  FT_SEARCH_ACC=0.5
  FT_SEARCH_ANG_SPD=3.0
  FT_SEARCH_ANG_ACC=10.0
  FT_SEARCH_RETRACT_ACC=10.0
  FT_SEARCH_RETRACT_SPD=3.0
  FT_SEARCH_RETRACT_M=0.002
  FT_SEARCH_RETRACT_RAD=d2r(4.25)
  ft_search_history_cntr=0
  def ft_trajectory_search_start(f3d=-1.0,t3d=-1.0):
  ft_select=ON_FALSE8D
  ft_limits=ON_ZERO8D
  ft_abs=ON_FALSE6D
  frameID=0
  frameRPY=ON_ZERO3D
  popupmsg=False
  speedLimit=0
  if(f3d>0):
  ft_select[6]=True
  ft_limits[6]=f3d
  end
  if(t3d>0):
  ft_select[7]=True
  ft_limits[7]=t3d
  end
  retVal=ft_limit_start(ft_select,ft_limits,ft_abs,speedLimit,frameID,frameRPY,popupmsg)
  cb_trajectory_return_validator(retVal,"F/T Limit: ")
  return retVal
  end
  def ft_trajectory_limited(trajectoryID,ft_select=ON_FALSE8D,ft_limits=ON_ZERO8D,ft_abs=ON_FALSE6D,frameID=0,frameRPY=ON_ZERO3D,isSearchReturn=False,popupmsg=True):
  speedLimit=0
  retVal=ft_limit_start(ft_select,ft_limits,ft_abs,speedLimit,frameID,frameRPY,popupmsg)
  cb_trajectory_return_validator(retVal,"F/T Limit: ")
  retVal=cb_trajectory(trajectoryID,isSearchReturn,popupmsg)
  ft_limit_stop()
  return retVal
  end
  def ft_trajectory_move_relative_limited_array(relativeOffsetsPoseArray=[ON_ZEROPOSE],ft_select=ON_FALSE8D,ft_limits=ON_ZERO8D,ft_abs=ON_FALSE6D,frameID=1,frameRPY=ON_ZERO3D,speed=0.05,acc=1.2,angularSpeed=3.0,angularAcc=10.0,isSearchReturn=False,popupmsg=True):
  local retVal=0
  frameRotVec=rpy2rotvec(frameRPY)
  frame6D=[0.0,0.0,0.0,frameRotVec[0],frameRotVec[1],frameRotVec[2]]
  frame=p[0.0,0.0,0.0,frameRotVec[0],frameRotVec[1],frameRotVec[2]]
  if((frameID%2)==1):
  startPose=get_actual_tcp_pose()
  startPose=pose_trans(startPose,frame)
  else:
  startPose=pose_trans(ON_ZEROPOSE,frame)
  end
  cb_trajectory_path_init(True,frameID,frame6D,speed,acc,angularSpeed,angularAcc)
  retVal=on_xmlrpc.cb_trajectory_waypoint([startPose[0]*1000.0,startPose[1]*1000.0,startPose[2]*1000.0,startPose[3],startPose[4],startPose[5]])
  cb_trajectory_return_validator(retVal,"OnWaypoint: ")
  cb_trajectory_waypoints_init(relativeOffsetsPoseArray,startPose,True,frameID)
  trajectoryID=cb_trajectory_path_init_end()
  retVal=ft_trajectory_limited(trajectoryID,ft_select,ft_limits,ft_abs,frameID,frameRPY,isSearchReturn,popupmsg)
  return retVal
  end
  def ft_trajectory_move_relative_limited(relativeOffsets=ON_ZEROPOSE,ft_select=ON_FALSE8D,ft_limits=ON_ZERO8D,ft_abs=ON_FALSE6D,frameID=1,frameRPY=ON_ZERO3D,speed=0.05,acc=1.2,angularSpeed=3.0,angularAcc=10.0,isSearchReturn=False,popupmsg=True):
  retVal=ft_trajectory_move_relative_limited_array([relativeOffsets],ft_select,ft_limits,ft_abs,frameID,frameRPY,speed,acc,angularSpeed,angularAcc,isSearchReturn,popupmsg)
  return retVal
  end
  def ft_trajectory_move_absolute_limited_array(fixPoseArray,ft_select=ON_FALSE8D,ft_limits=ON_ZERO8D,ft_abs=ON_FALSE6D,speed=0.05,acc=1.2,angularSpeed=3.0,angularAcc=10.0,isSearchReturn=False,popupmsg=True):
  local retVal=0
  frame6D=ON_ZERO6D
  frameID=0
  frameRPY=ON_ZERO3D
  local startPose=ON_ZEROPOSE
  cb_trajectory_path_init(False,frameID,frame6D,speed,acc,angularSpeed,angularAcc)
  cb_trajectory_waypoints_init(fixPoseArray,startPose,False,frameID)
  trajectoryID=cb_trajectory_path_init_end()
  retVal=ft_trajectory_limited(trajectoryID,ft_select,ft_limits,ft_abs,frameID,frameRPY,isSearchReturn,popupmsg)
  return retVal
  end
  def ft_trajectory_move_absolute_limited(fixPose,ft_select=ON_FALSE8D,ft_limits=ON_ZERO8D,ft_abs=ON_FALSE6D,speed=0.05,acc=1.2,angularSpeed=3.0,angularAcc=10.0,isSearchReturn=False,popupmsg=True):
  retVal=ft_trajectory_move_absolute_limited_array([fixPose],ft_select,ft_limits,ft_abs,speed,acc,angularSpeed,angularAcc,isSearchReturn,popupmsg)
  return retVal
  end
  def ft_search_relativeZ(tool_index,searchDistZ,speed=0.03,forceZ=5.0,popupmsg=True):
  on_tcp_set_actual_to(tool_index!=ON_DI_SECONDARY)
  ft_select=ON_FALSE8D
  ft_select[2]=True
  ft_limits=ON_ZERO8D
  ft_limits[2]=forceZ
  ft_abs=ON_FALSE6D
  frameID=1
  frameRPY=ON_ZERO3D
  searchUntil=ON_ZEROPOSE
  searchUntil[2]=searchDistZ
  isSearchReturn=True
  local retVal=ft_trajectory_move_relative_limited(searchUntil,ft_select,ft_limits,ft_abs,frameID,frameRPY,speed,FT_SEARCH_ACC,FT_SEARCH_ANG_SPD,FT_SEARCH_ANG_ACC,isSearchReturn,popupmsg)
  return retVal
  end
  def ft_search_get_retract_pose(poseArray,actualStep,retract_m=-1,retract_rad=-1):
  local SafeIndex=actualStep+1
  if SafeIndex>=FT_SEARCH_HISTORY_LENGTH:
  SafeIndex=0
  end
  local actualPose=poseArray[actualStep]
  local safePose=poseArray[SafeIndex]
  local directionPose=pose_trans(pose_inv(actualPose),safePose)
  local directionUnit=normalize([directionPose[0],directionPose[1],directionPose[2],directionPose[3],directionPose[4],directionPose[5]])
  local Pdist=pose_dist(actualPose,safePose)
  local retractVector=directionPose
  if(retract_m>=0):
  retractVector[0]=directionUnit[0]*retract_m
  retractVector[1]=directionUnit[1]*retract_m
  retractVector[2]=directionUnit[2]*retract_m
  end
  if(retract_rad>=0):
  retractVector[3]=directionUnit[3]*retract_rad
  retractVector[4]=directionUnit[4]*retract_rad
  retractVector[5]=directionUnit[5]*retract_rad
  end
  ft_search_safe_pose=pose_trans(actualPose,retractVector)
  return ft_search_safe_pose
  end
  thread ft_search_safety_thread():
  ft_search_abscntr=0
  ft_search_history_cntr=0
  while True:
  enter_critical
  ft_search_abscntr=ft_search_abscntr+1
  ft_search_history_cntr=ft_search_history_cntr+1
  if ft_search_history_cntr>=FT_SEARCH_HISTORY_LENGTH:
  ft_search_history_cntr=0
  end
  ft_search_history[ft_search_history_cntr]=get_actual_tcp_pose()
  exit_critical
  sync()
  end
  end
  ft_search_safety_thrd=run ft_search_safety_thread()
  def ft_search_retract(retractPose):
  if(on_speedl_integer_get()==0):
  movel(retractPose,a=FT_SEARCH_ACC,v=FT_SEARCH_RETRACT_SPD)
  else:
  cb_trajectory_move_absolute(retractPose,FT_SEARCH_RETRACT_SPD,FT_SEARCH_ACC,(FT_SEARCH_RETRACT_SPD*4.0),(FT_SEARCH_ACC*4.0),False)
  end
  end
  def ft_search_OK_retract(retractPose):
  if ft_search_return==0:
  ft_search_retract(retractPose)
  end
  end

  #======    End of OnRobot FT Trajectory    ======#
  #======    OnRobot FT Trajectory Spiral    ======#

  def cb_trajectory_spiral(spiralStartEndPoses=[ON_ZEROPOSE,ON_ZEROPOSE],isRelative=True,speed=0.05,acc=1.2,angularSpeed=3.0,angularAcc=10.0,increase=0.001,direction=False,closingCircle=False,popupmsg=True):
  local retVal=0
  local isSearchReturn=False
  trajectoryID=cb_trajectory_spiral_init(spiralStartEndPoses,isRelative,speed,acc,angularSpeed,angularAcc,increase,direction,closingCircle)
  retVal=cb_trajectory(trajectoryID,isSearchReturn,popupmsg)
  return retVal
  end
  def cb_trajectory_spiral_limited(spiralStartEndPoses=[ON_ZEROPOSE,ON_ZEROPOSE],ft_select=ON_FALSE8D,ft_limits=ON_ZERO8D,ft_abs=ON_FALSE6D,isRelative=True,speed=0.05,acc=1.2,angularSpeed=3.0,angularAcc=10.0,increase=0.01,direction=False,closingCircle=False,isSearchReturn=False,popupmsg=True):
  local retVal=0
  local frameRPY=ON_ZERO3D
  local frameID=1
  trajectoryID=cb_trajectory_spiral_init(spiralStartEndPoses,isRelative,speed,acc,angularSpeed,angularAcc,increase,direction,closingCircle)
  retVal=ft_trajectory_limited(trajectoryID,ft_select,ft_limits,ft_abs,frameID,frameRPY,isSearchReturn,popupmsg)
  return retVal
  end

  #======    End of OnRobot FT Trajectory Spiral    ======#
  #======    OnRobot FT Insert Part Messages    ======#

  ft_insert_part_error_title="OnRobot - Insert Part error"
  ft_insert_part_state_error_start="Wrong F/T Insert Part status when initializing.<br>Another thread is using an F/T Insert Part command. Program halted."
  ft_insert_part_state_error_return="Wrong F/T Insert Part status when returning.<br>Another thread is using an F/T Insert Part command. Program halted."
  ft_insert_part_return_title="OnRobot - Insert Part"
  ft_insert_part_return_0="The insertion has reached the maximal insertion depth."
  ft_insert_part_return_1="The insertion bumped after the minimal insertion depth."
  ft_insert_part_return_2="The insertion slowed down after the minimal insertion depth."
  ft_insert_part_return_3="The insertion got stuck before the minimal insertion depth."
  ft_insert_part_return_4="The command has timed out after the minimal insertion depth."
  ft_insert_part_return_5="The command has timed out before the minimal insertion depth."
  ft_insert_part_return_6="The side-force/-torque limit has been reached after the minimal insertion depth."
  ft_insert_part_return_7="The side-force/-torque limit has been reached before the minimal insertion depth."
  ft_insert_part_return_8="Parameter error returned from the Compute Box.<br>Check the parameters for the F/T Insert Part command."
  ft_insert_part_return_unknown="F/T Insert Part finished with unknown return value."

  #======    End of OnRobot FT Insert Part Messages    ======#
  #======    OnRobot FT Insert Part    ======#

  ft_insert_part_state=0
  ft_insert_part_return=0
  ft_sensor_filter_insertpart_hex=6
  ft_insert_part_frameID=1
  ft_insert_part_frameID_default=1
  ft_insert_part_frameRPY=ON_ZERO3D
  ft_insert_part_frameRPY_default=ON_ZERO3D
  ft_insert_part_retAccept=[True,True,True,False,False,False,False,False,False]
  ft_insert_part_retAccept_default=[True,True,True,False,False,False,False,False,False]
  FT_INSERT_PART_STATE_IDLE=0
  FT_INSERT_PART_STATE_INIT=1
  FT_INSERT_PART_STATE_STARTED=2
  FT_INSERT_PART_STATE_RETURNING=3
  ft__insert_part_param_error_minDistZ="Please define parameter 'minDistZ' as a positive real number in meters!"
  ft__insert_part_param_error_forceZ="Please define parameter 'forceZ' as a positive number in Newtons!"
  ft__insert_part_param_error_maxDistZ="Please define parameter 'maxDistZ' as a positive real number in meters!"
  ft__insert_part_param_error_maxDistZ_minDistZ="Please define the parameters as 'maxDistZ' >= 'minDistZ'!"
  ft__insert_part_param_error_expSpeed="Please define parameter 'expSpeed' as a positive real number in meters!"
  ft__insert_part_param_error_deltaForce="Please define parameter 'deltaForce' as a positive number in Newtons!"
  ft__insert_part_param_error_timeOut="Please define parameter 'timeOut' as a positive number in seconds!"
  ft__insert_part_param_error_FTLimits="Please define parameter 'FTLimits' as a 6-element array of positive numbers in Newtons & Newton-meters!"
  ft__insert_part_param_error_PGainFxy="Please define parameter 'PGainFxy' as a positive real number!"
  ft__insert_part_param_error_PGainFz="Please define parameter 'PGainFz' as a positive real number!"
  ft__insert_part_param_error_PGainTxy="Please define parameter 'PGainTxy' as a positive real number!"
  ft__insert_part_param_error_PGainTz="Please define parameter 'PGainTz' as a positive real number!"
  def ft_insert_part(forceZ,minDistZ,maxDistZ=0.0,deltaForce=0.0,expSpeed=0.0,timeOut=0,compliance=[True,True,True,True,True,True],FTLimits=ON_ZERO6D,PGainFxy=1.0,PGainFz=1.0,PGainTxy=0.2,PGainTz=0.2,popupmsg=True):
  sync()
  if ON_DEBUG_LOG:
  textmsg("Insert Part starting..")
  end
  if not(ft_insert_part_state==FT_INSERT_PART_STATE_IDLE):
  textmsg("ft_insert_part_state: ",ft_insert_part_state)
  popup(ft_insert_part_state_error_start,title=ft_insert_part_error_title,error=True,blocking=False)
  halt
  else:
  enter_critical
  ft_insert_part_state=FT_INSERT_PART_STATE_INIT
  exit_critical
  end
  ft_insert_part_return=0
  if not(minDistZ>=0):
  ft_insert_part_return=8
  popup(ft__insert_part_param_error_minDistZ,title=ft_insert_part_error_title,error=True,blocking=True)
  elif not(forceZ!=0):
  ft_insert_part_return=8
  popup(ft__insert_part_param_error_forceZ,title=ft_insert_part_error_title,error=True,blocking=True)
  elif not(maxDistZ>=0):
  ft_insert_part_return=8
  popup(ft__insert_part_param_error_maxDistZ,title=ft_insert_part_error_title,error=True,blocking=False)
  elif not(maxDistZ>=minDistZ or maxDistZ==0):
  ft_insert_part_return=8
  popup(ft__insert_part_param_error_maxDistZ_minDistZ,title=ft_insert_part_error_title,error=True,blocking=False)
  elif not(expSpeed>=0):
  ft_insert_part_return=8
  popup(ft__insert_part_param_error_expSpeed,title=ft_insert_part_error_title,error=True,blocking=False)
  elif not(deltaForce>=0):
  ft_insert_part_return=8
  popup(ft__insert_part_param_error_deltaForce,title=ft_insert_part_error_title,error=True,blocking=False)
  elif not(timeOut>=0):
  ft_insert_part_return=8
  popup(ft__insert_part_param_error_timeOut,title=ft_insert_part_error_title,error=True,blocking=False)
  elif not(FTLimits[0]>=0):
  ft_insert_part_return=8
  popup(ft__insert_part_param_error_FTLimits,title=ft_insert_part_error_title,error=True,blocking=False)
  elif not(FTLimits[1]>=0):
  ft_insert_part_return=8
  popup(ft__insert_part_param_error_FTLimits,title=ft_insert_part_error_title,error=True,blocking=False)
  elif not(FTLimits[3]>=0):
  ft_insert_part_return=8
  popup(ft__insert_part_param_error_FTLimits,title=ft_insert_part_error_title,error=True,blocking=False)
  elif not(FTLimits[4]>=0):
  ft_insert_part_return=8
  popup(ft__insert_part_param_error_FTLimits,title=ft_insert_part_error_title,error=True,blocking=False)
  elif not(FTLimits[5]>=0):
  ft_insert_part_return=8
  popup(ft__insert_part_param_error_FTLimits,title=ft_insert_part_error_title,error=True,blocking=False)
  elif not(PGainFxy>0):
  ft_insert_part_return=8
  popup(ft__insert_part_param_error_PGainFxy,title=ft_insert_part_error_title,error=True,blocking=False)
  elif not(PGainFz>0):
  ft_insert_part_return=8
  popup(ft__insert_part_param_error_PGainFz,title=ft_insert_part_error_title,error=True,blocking=False)
  elif not(PGainTxy>0):
  ft_insert_part_return=8
  popup(ft__insert_part_param_error_PGainTxy,title=ft_insert_part_error_title,error=True,blocking=False)
  elif not(PGainTz>0):
  ft_insert_part_return=8
  popup(ft__insert_part_param_error_PGainTz,title=ft_insert_part_error_title,error=True,blocking=False)
  end
  if(ft_insert_part_return!=0):
  halt
  end
  on_tcp_offset_send(get_tcp_offset())
  local retAccept=ft_insert_part_retAccept
  ft_insert_part_retAccept=ft_insert_part_retAccept_default
  local ft_compliance=compliance
  ft_compliance[2]=True
  local ft_threshold=[FTLimits[0],FTLimits[1],(forceZ+deltaForce),FTLimits[3],FTLimits[4],FTLimits[5]]
  i=0
  while i<6:
  if ft_compliance[i]:
  ft_threshold[i]=0
  end
  i=i+1
  end
  local flags=binary_list_to_integer(ft_compliance)+(ft_insert_part_frameID*64)
  ft_insert_part_frameID=ft_insert_part_frameID_default
  local ft_insert_part_frame=rpy2rotvec(ft_insert_part_frameRPY)
  ft_insert_part_frameRPY=ft_insert_part_frameRPY_default
  sync()
  ft_insert_part_return=ft_pin_insertion(minDistZ,forceZ,compliance,maxDistZ,expSpeed,deltaForce,timeOut,FTLimits,PGainFxy,PGainFz,PGainTxy,PGainTz)
  if ON_DEBUG_LOG:
  textmsg("Insert Part returned.")
  end
  if ft_insert_part_return==0:
  if(popupmsg and(not retAccept[0])):
  popup(ft_insert_part_return_0,title=ft_insert_part_return_title,warning=True,blocking=True)
  end
  elif ft_insert_part_return==1:
  if(popupmsg and(not retAccept[1])):
  popup(ft_insert_part_return_1,title=ft_insert_part_return_title,warning=True,blocking=True)
  end
  elif ft_insert_part_return==2:
  if(popupmsg and(not retAccept[2])):
  popup(ft_insert_part_return_2,title=ft_insert_part_return_title,warning=True,blocking=True)
  end
  elif ft_insert_part_return==3:
  if(popupmsg and(not retAccept[3])):
  popup(ft_insert_part_return_3,title=ft_insert_part_return_title,warning=True,blocking=True)
  end
  elif ft_insert_part_return==4:
  if(popupmsg and(not retAccept[4])):
  popup(ft_insert_part_return_4,title=ft_insert_part_return_title,warning=True,blocking=True)
  end
  elif ft_insert_part_return==5:
  if(popupmsg and(not retAccept[5])):
  popup(ft_insert_part_return_5,title=ft_insert_part_return_title,warning=True,blocking=True)
  end
  elif ft_insert_part_return==6:
  if(popupmsg and(not retAccept[6])):
  popup(ft_insert_part_return_6,title=ft_insert_part_return_title,warning=True,blocking=True)
  end
  elif ft_insert_part_return==7:
  if(popupmsg and(not retAccept[7])):
  popup(ft_insert_part_return_7,title=ft_insert_part_return_title,warning=True,blocking=True)
  end
  else:
  popup(ft_insert_part_return_unknown,title=ft_insert_part_return_title,warning=True,blocking=True)
  end
  enter_critical
  ft_insert_part_state=FT_INSERT_PART_STATE_IDLE
  exit_critical
  if ON_DEBUG_LOG:
  textmsg("End of Insert Part.")
  end
  return ft_insert_part_return
  end
  ft_peakFzScanner_flag=False
  ft_abs_Fz=0
  ft_abs0_Fz=False
  thread ft_peakFzScanner():
  ft_peakFzScanner_flag=True
  ft_abs_Fz=0
  while(ft_peakFzScanner_flag==True):
  local norm_Fz=norm(FT_Tool[2])
  if(ft_abs0_Fz):
  ft_abs_Fz=0
  ft_abs0_Fz=False
  elif(ft_abs_Fz<norm_Fz):
  ft_abs_Fz=norm_Fz
  end
  sync()
  end
  end
  ft_fpid_i_pin=0.0
  ft_fpid_d_pin=0.0
  ft_fpid_i_pin_default=0.0
  ft_fpid_d_pin_default=0.0
  ft_tpid_i_pin=0.0
  ft_tpid_d_pin=0.0
  ft_tpid_i_pin_default=0.0
  ft_tpid_d_pin_default=0.0
  def ft_pin_insertion(minDistZ,forceZ,compliance=[True,True,True,True,True,True],maxDistZ=0,expSpeed=0,deltaForce=1,timeOut=0,FTLimits=[999,999,0,999,999,999],PGainFxy=1.0,PGainFz=1.0,PGainTxy=0.2,PGainTz=0.2):
  sync()
  local pinRet=0
  local frameID=1
  local startPose=get_actual_tcp_pose()
  if maxDistZ==0:
  maxDistZ=minDistZ
  end
  local dist2Reach=maxDistZ
  sync()
  local selectThreshold=[False,False,False,False,False,False]
  local ft_select=compliance
  ft_select[2]=True
  local ft_values=[0.0,0.0,0.0,0.0,0.0,0.0]
  ft_values[2]=forceZ+0.0
  local i=0
  while(i<6):
  selectThreshold[i]=not(ft_select[i])
  i=i+1
  end
  local pin_useTimeOut=True
  if timeOut==0:
  pin_useTimeOut=False
  end
  local timeOut100ms=timeOut*10
  local deltaD=expSpeed/10
  ft_pin_currentDist=0
  local peakScanner=run ft_peakFzScanner()
  sync()
  local pin_gainP=[PGainFxy,PGainFxy,PGainFz,PGainTxy,PGainTxy,PGainTz]
  local pin_gainI=[ft_fpid_i_pin,ft_fpid_i_pin,ft_fpid_i_pin,ft_tpid_i_pin,ft_tpid_i_pin,ft_tpid_i_pin]
  local pin_gainD=[ft_fpid_d_pin,ft_fpid_d_pin,ft_fpid_d_pin,ft_tpid_d_pin,ft_tpid_d_pin,ft_tpid_d_pin]
  if on_hex:
  on_xmlrpc.ft_sensor_filter(ft_sensor_filter_insertpart_hex)
  end
  pin_speed_variation=0.0
  pin_keep_force=-1.0
  pin_auto_keep_force=False
  pin_keep_torque=-1.0
  pin_auto_keep_torque=False
  ft_ftcontrol_start(ft_select=ft_select,ft_values=ft_values,frameID=frameID,frameRPY=[0,0,0],gainP=pin_gainP,gainI=pin_gainI,gainD=pin_gainD,speed_variation=pin_speed_variation,keep_force=pin_keep_force,auto_keep_force=pin_auto_keep_force,keep_torque=pin_keep_torque,auto_keep_torque=pin_auto_keep_torque)
  local cntr=0
  local leaveInsertion=False
  local bumpZeroPeak=True
  local pin_actual_pose=get_actual_tcp_pose()
  ft_pin_currentDist=point_dist(startPose,pin_actual_pose)
  local pin_last_pose=pin_actual_pose
  ft_actual_deltaD=deltaD
  while((ft_pin_currentDist<dist2Reach)and not leaveInsertion):
  on_wait_ms(100)
  pin_actual_pose=get_actual_tcp_pose()
  ft_pin_currentDist=point_dist(startPose,pin_actual_pose)
  ft_actual_deltaD=(ft_actual_deltaD+pose_dist(pin_last_pose,pin_actual_pose))/2
  if(ft_threshold_check(FTLimits,selectThreshold,True)):
  leaveInsertion=True
  if(ft_pin_currentDist<minDistZ):
  pinRet=7
  else:
  pinRet=6
  end
  ft_ftcontrol_stop()
  elif(pin_useTimeOut and(cntr>timeOut100ms)):
  leaveInsertion=True
  if(ft_pin_currentDist<minDistZ):
  pinRet=5
  else:
  pinRet=4
  end
  ft_ftcontrol_stop()
  elif(ft_actual_deltaD<deltaD and cntr>=10):
  leaveInsertion=True
  if(ft_pin_currentDist<minDistZ):
  pinRet=3
  ft_ftcontrol_stop()
  else:
  pinRet=2
  end
  elif(ft_pin_currentDist>=minDistZ):
  if bumpZeroPeak:
  bumpZeroPeak=False
  ft_abs0_Fz=True
  sync()
  else:
  if(ft_abs_Fz>norm(forceZ+deltaForce)and not ft_abs0_Fz):
  ft_peakFzScanner_flag=False
  leaveInsertion=True
  pinRet=1
  end
  end
  end
  pin_last_pose=pin_actual_pose
  cntr=cntr+1
  sync()
  end
  ft_ftcontrol_stop()
  on_xmlrpc.ft_sensor_filter(FT_SENSOR_FILTER_DEFAULT)
  ft_peakFzScanner_flag=False
  kill peakScanner
  ft_fpid_i_pin=ft_fpid_i_pin_default
  ft_fpid_d_pin=ft_fpid_d_pin_default
  ft_tpid_i_pin=ft_tpid_i_pin_default
  ft_tpid_d_pin=ft_tpid_d_pin_default
  return pinRet
  end

  #======    End of OnRobot FT Insert Part    ======#
  #======    OnRobot FT Search Part
    ======#

  def hex_search_part(frameID,axis,isDirectionPositive,max_dist,contact_ft,tcp_speed,retraction):
  relativeOffsets=ON_ZEROPOSE
  ft_select=ON_FALSE8D
  ft_limits=ON_ZERO8D
  ft_abs=ON_FALSE6D
  frameRPY=ON_ZERO3D
  if axis<3:
  speed=tcp_speed
  angularSpeed=tcp_speed*4
  elif axis>2:
  speed=tcp_speed/4
  angularSpeed=tcp_speed
  end
  angularAcc=9.0
  acc=0.6
  isSearchReturn=True
  popupmsg=False
  ft_select[axis]=True
  if isDirectionPositive==True:
  d=1.0
  elif isDirectionPositive==False:
  d=-1.0
  end
  relativeOffsets[axis]=d*max_dist
  ft_limits[axis]=d*contact_ft
  if axis>2 and relativeOffsets[axis]>d2r(179)or relativeOffsets[axis]<-d2r(179):
  if relativeOffsets[axis]>d2r(360):
  relativeOffsets[axis]=d2r(360)/3
  elif relativeOffsets[axis]<-d2r(360):
  relativeOffsets[axis]=-d2r(360)/3
  else:
  relativeOffsets[axis]=relativeOffsets[axis]/3
  end
  relativeOffsetsPoseArray=[relativeOffsets,relativeOffsets,relativeOffsets]
  else:
  relativeOffsetsPoseArray=[relativeOffsets,ON_ZEROPOSE,ON_ZEROPOSE]
  end
  search_return=ft_trajectory_move_relative_limited_array(relativeOffsetsPoseArray,ft_select,ft_limits,ft_abs,frameID,frameRPY,speed,acc,angularSpeed,angularAcc,isSearchReturn,popupmsg)
  if search_return<0:
  ft_search_return=search_return
  return ft_search_return
  end
  if retraction==True and frameID==1:
  if axis<3:
  relativeOffsets[axis]=-d*0.002
  elif axis>2:
  relativeOffsets[axis]=-d*d2r(2)
  end
  movel(pose_trans(get_actual_tcp_pose(),relativeOffsets),a=0.5,v=speed,t=0,r=0)
  elif retraction==True and frameID==0:
  retract_pose=get_actual_tcp_pose()
  if axis<3:
  retract_pose[axis]=retract_pose[axis]-d*0.002
  elif axis>2:
  retract_angle=ON_ZEROPOSE
  retract_angle[axis]=-d*d2r(2)
  retract_pose=pose_add(retract_angle,retract_pose)
  end
  movel(retract_pose,a=0.5,v=speed,t=0,r=0)
  end
  ft_search_return=0
  return ft_search_return
  end
  def HEX_Search_NOK():
  return(ft_search_return!=0)
  end

  #======    End of OnRobot FT Search Part
    ======#
  #======    OnRobot FT Search Center    ======#

  hex_center_pose=ON_ZEROPOSE
  hex_center_distances=[0.0,0.0,0.0,0.0,0.0,0.0]
  def hex_centering_1D(axis,frameID,max_dist,tcp_speed,contact_ft):
  relativeOffsets=ON_ZEROPOSE
  ft_select=ON_FALSE8D
  ft_limits=ON_ZERO8D
  ft_abs=ON_FALSE6D
  frameRPY=ON_ZERO3D
  if axis<3:
  speed=tcp_speed
  angularSpeed=tcp_speed*4
  elif axis>2:
  speed=tcp_speed/4
  angularSpeed=tcp_speed
  end
  angularAcc=9.0
  acc=0.6
  isSearchReturn=True
  popupmsg=False
  relativeOffsets[axis]=max_dist
  if axis>2 and relativeOffsets[axis]>d2r(179):
  rotational_180=True
  if relativeOffsets[axis]>d2r(360):
  relativeOffsets[axis]=d2r(360)/3
  else:
  relativeOffsets[axis]=relativeOffsets[axis]/3
  end
  relativeOffsetsPoseArray=[relativeOffsets,relativeOffsets,relativeOffsets]
  else:
  rotational_180=False
  relativeOffsetsPoseArray=[relativeOffsets,ON_ZEROPOSE,ON_ZEROPOSE]
  end
  ft_select[axis]=True
  ft_limits[axis]=contact_ft
  start_pose=get_actual_tcp_pose()
  ft_bias()
  search_return=ft_trajectory_move_relative_limited_array(relativeOffsetsPoseArray,ft_select,ft_limits,ft_abs,frameID,frameRPY,speed,acc,angularSpeed,angularAcc,isSearchReturn,popupmsg)
  if search_return<0 and rotational_180==True:
  relativeOffsets[axis]=-relativeOffsets[axis]
  relativeOffsetsPoseArray=[relativeOffsets,relativeOffsets,relativeOffsets]
  cb_trajectory_move_relative_array(relativeOffsetsPoseArray,frameID,frameRPY,speed,acc,angularSpeed,angularAcc,popupmsg)
  return-1
  elif search_return<0 and rotational_180==False:
  movel(start_pose,a=0.5,v=speed,t=0,r=0)
  return-1
  end
  sleep(0.2)
  pose_1=get_actual_tcp_pose()
  if axis<3:
  dist_pose1=pose_dist(pose_1,start_pose)
  dist_pose=dist_pose1
  elif axis>2:
  pose_1s=pose_trans(pose_inv(start_pose),pose_1)
  sub_poses=pose_sub(pose_1s,ON_ZEROPOSE)
  angle_dist1=sub_poses[axis]
  if angle_dist1<0:
  angle_dist1=angle_dist1+d2r(360)
  end
  dist_pose=angle_dist1
  end
  relativeOffsets[axis]=-max_dist-dist_pose
  ft_limits[axis]=-contact_ft
  if axis>2 and relativeOffsets[axis]<-d2r(179):
  rotational_180=True
  if relativeOffsets[axis]<-d2r(360):
  relativeOffsets[axis]=-d2r(360)/3
  else:
  relativeOffsets[axis]=relativeOffsets[axis]/3
  end
  relativeOffsetsPoseArray=[relativeOffsets,relativeOffsets,relativeOffsets]
  else:
  rotational_180=False
  relativeOffsetsPoseArray=[relativeOffsets,ON_ZEROPOSE,ON_ZEROPOSE]
  end
  search_return=ft_trajectory_move_relative_limited_array(relativeOffsetsPoseArray,ft_select,ft_limits,ft_abs,frameID,frameRPY,speed,acc,angularSpeed,angularAcc,isSearchReturn,popupmsg)
  if search_return<0 and rotational_180==True:
  relativeOffsets[axis]=(-relativeOffsets[axis]*3-dist_pose)/3
  relativeOffsetsPoseArray=[relativeOffsets,relativeOffsets,relativeOffsets]
  cb_trajectory_move_relative_array(relativeOffsetsPoseArray,frameID,frameRPY,speed,acc,angularSpeed,angularAcc,popupmsg)
  return-2
  elif search_return<0 and rotational_180==False:
  movel(start_pose,a=0.5,v=speed,t=0,r=0)
  return-2
  end
  sleep(0.2)
  pose_2=get_actual_tcp_pose()
  if axis<3:
  hex_center_distance=pose_dist(pose_1,pose_2)/2
  hex_center_pose=interpolate_pose(pose_1,pose_2,0.5)
  elif axis>2:
  pose_2s=pose_trans(pose_inv(start_pose),pose_2)
  sub_poses=pose_sub(pose_2s,pose_1s)
  hex_center_pose=interpolate_pose(pose_2,pose_1,0.5)
  if sub_poses[axis]>0:
  angle_offset=ON_ZEROPOSE
  angle_offset[axis]=d2r(180)
  hex_center_pose=pose_trans(hex_center_pose,angle_offset)
  end
  sub_poses=pose_sub(pose_1s,pose_trans(pose_inv(start_pose),hex_center_pose))
  hex_center_distance=sub_poses[axis]
  end
  movel(hex_center_pose,a=0.5,v=speed,t=0,r=0)
  hex_center_distances[axis]=hex_center_distance
  return 0
  end
  def hex_centering(CIA,frameID,max_dist,tcp_speed,contact_ft):
  translational=False
  rotational=False
  l=length(CIA)
  i=0
  while i<l:
  if CIA[i]<3:
  translational=True
  elif CIA[i]>2:
  rotational=True
  end
  if translational==True and rotational==True:
  return-10
  end
  i=i+1
  end
  i=0
  while i<l:
  axis=CIA[i]
  centering_return=hex_centering_1D(axis,frameID,max_dist,tcp_speed,contact_ft)
  if centering_return<0:
  ft_search_return=centering_return-i*2
  return ft_search_return
  end
  i=i+1
  end
  ft_search_return=0
  return ft_search_return
  end

  #======    End of OnRobot FT Search Center    ======#

  #======    End of OnRobot RG2-FT Proximity AVG Messages    ======#
  #======    OnRobot RG2-FT Proximity AVG    ======#

  rg2ft_proxi_avg_window_default=10
  rg2ft_proxi_avg_window=10
  rg2ft_proxi_avg_window_last=rg2ft_proxi_avg_window
  rg2ft__proxi_avg_window_error_title="OnRobot - Gripper Proximity"
  rg2ft__proxi_avg_window_error_windowSize="Please define parameter windowSize as a positive integer between 0 and 20."
  def rg2ft_proxi_avg_window_set(windowSize=10):
  sync()
  if ON_DEBUG_LOG:
  textmsg("Gripper Proxi Avg Window Set command starting..")
  end
  windowSize=floor(windowSize+0.5)
  if not(windowSize>0 and windowSize<=20):
  popup(rg2ft__proxi_avg_window_error_windowSize,title=rg2ft__proxi_avg_window_error_title,error=True,blocking=False)
  halt
  end
  rg2ft_proxi_avg_window_last=rg2ft_proxi_avg_window
  rg2ft_proxi_avg_window=windowSize
  on_xmlrpc.rg2ft_proxi_avg(windowSize)
  if ON_DEBUG_LOG:
  textmsg("Gripper Proxi Avg Window Set command ended.")
  end
  end
  def rg2ft_proxi_avg_window_reset_last():
  rg2ft_proxi_avg_window_set(rg2ft_proxi_avg_window_last)
  end
  def rg2ft_proxi_avg_window_reset_default():
  rg2ft_proxi_avg_window_set(rg2ft_proxi_avg_window_default)
  end

  #======    End of OnRobot RG2-FT Proximity AVG    ======#

  #======    End of OnRobot RG2-FT Width Filter Messages    ======#
  #======    OnRobot RG2-FT Width Filter    ======#

  rg2ft_width_filter=10
  rg2ft__width_filter_error_title="OnRobot - Gripper Proximity"
  rg2ft__width_filter_error_bufferSize="Please define parameter bufferSize as a positive integer between 0 and 20."
  def rg2ft_width_filter_set(bufferSize=10):
  sync()
  if ON_DEBUG_LOG:
  textmsg("Gripper Width filtering set command starting..")
  end
  bufferSize=floor(bufferSize+0.5)
  if not(bufferSize>0 and bufferSize<=20):
  popup(rg2ft__width_filter_error_bufferSize,title=rg2ft__width_filter_error_title,error=True,blocking=False)
  halt
  end
  rg2ft_width_filter=bufferSize
  on_xmlrpc.rg2ft_width_filter(bufferSize)
  if ON_DEBUG_LOG:
  textmsg("Gripper Width filtering set command stopping..")
  end
  end

  #======    End of OnRobot RG2-FT Width Filter    ======#
  # end: URCap Installation Node
  step_count_fe5c8550_9ec4_4cb7_ae6b_a9e4c63ad615 = 0.0
  thread Step_Counter_Thread_62d5d6ae_bf13_4d68_84ae_8bc3a7324278():
    while (True):
      step_count_fe5c8550_9ec4_4cb7_ae6b_a9e4c63ad615 = step_count_fe5c8550_9ec4_4cb7_ae6b_a9e4c63ad615 + 1.0
      sync()
    end
  end
  run Step_Counter_Thread_62d5d6ae_bf13_4d68_84ae_8bc3a7324278()
  $ 1 "Robot Program"
  # begin: URCap Program Node
  #   Source: OnRobot, 5.3.2, OnRobot A/S
  #   Type: RG2-FT Grip
  $ 2 "RG2-FT Grip"
on_return = rg2ft_grip(97.1, 40.0, tool_index = 0, blocking = True, depth_comp = False, popupmsg = True)
rg2ft_payload_set(mass = 0.0, tool_index = 0, use_guard = True)
  # end: URCap Program Node
end
